PROGRAM FunctionsAndFunctionBlocks

END_PROGRAM

(* stored: Version 1.1.0.1
   POU FunctionsAndFunctionBlocks: Id {b5f823cc-f761-4488-9157-3d2695b6a23f}, SpecialFunc None *)
